{attribute 'GeneratedUsingTerminal: EL2521-0000-1017'}
{attribute addProperty BoxType "EL2521-0000-1017"}
{attribute addProperty Id "ControlAT %Q*Control_DAEE1D523Frequency_valueAT %Q*UINT2"}
{attribute addProperty CRC "2458384612"}
{attribute addProperty Size "5"}
TYPE PTO_Control_9287F8E4 :
STRUCT
	{attribute addProperty Name "Control"}
	Control AT %Q* : Control_DAEE1D52;
	{attribute addProperty Name "Frequency_value"}
	Frequency_value AT %Q* : UINT;
END_STRUCT
END_TYPE

(* stored: Version 1.2.0.0, ProductVersion 3.1.4024.9
   DUT PTO_Control_9287F8E4: Id {ce3b25b1-d54c-4030-a7e9-1c7efb2cc532} *)
